// TIA Portal V20 export
TYPE "LAxisCtrl_typeTorqueLimiting"
TITLE = LAxisCtrl_typeTorqueLimiting
// Support: tech.team.motioncontrol@siemens.com 
// Fax: +49 (0) 9131/98-1297
   STRUCT
      limit : LReal := -1.0;   // Value of force/torque limiting (in the configured unit of measurement)
      mode : DInt := 0;   // 0: Force/Torque limiting; 1: Fixed stop detection
   END_STRUCT;
END_TYPE
